# EPICS substitutions: tpmacApp/pmc/xf10ida-mc02-plc05-cpu.substitutions
file "PLC_cpu_load.pmc"
{
pattern
{ PLC }
{ 5   }
}
